SUBAPPLICATION Ventilsteuerung (* Subapplication Type *)
  (* Standard: 61499-2 *)
  (* Version 1.0, 2025-01-31, franz *)
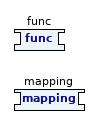
  SUBAPPS
    func : func;
    mapping : mapping;
  END_SUBAPPS
END_SUBAPPLICATION
